(* CODESYS project Mahle_FilterLine_TempControl_02_08_20.project
   Title: Mahle_FilterLine_TempControl_03_01_20
   Version: 0.0.0.0

Project tree, tasks and I/O mapping:
  MyController : TM218LDAE24DRHN, Schneider Electric, order no. TM218LDAE24DRHN, version 4.0.1.26
      settings: Expansion Tasks.Expansion 1 Task Name = 'MAST'; Expansion Tasks.Expansion 2 Task Name = 'MAST'
    application Application
      libraries: Standard, * (System)
      task MAST (cyclic, interval 20 ms, priority 15, watchdog 100 ms x 1) calls POU, POU_MC2
      function HiddenPOU [ST]
      global variables GVL
      program POU [FBD]
      function block tempAvergaging [ST]
      function block tempController [ST]
      function block calculateCycleTime [ST]
      function CheckBounds [ST]
      function block pressureAlarm [ST]
      program POU_MC2 [FBD]
    Embedded Functions
      IO : IO, Schneider Electric, version 4.0.1.26
          input  iwIO_IW0 : WORD  // IW0
          input  iAuto : BOOL  // IW0.I0
          input  iThyristorTrip2 : BOOL  // IW0.I1
          input  iStartPB : BOOL  // IW0.I2
          input  iStopPB : BOOL  // IW0.I3
          input  iStartPB2 : BOOL  // IW0.I4
          input  iStopPB2 : BOOL  // IW0.I5
          input  iThyristorTrip : BOOL  // IW0.I6
          input  iFwdSensor2 : BOOL  // IW0.I7
          input  iFwdSensor : BOOL  // IW0.I8
          input  iSafetyGuard : BOOL  // IW0.I10
          input  iSafetyGuard2 : BOOL  // IW0.I11
          input  iPanelPB : BOOL  // IW0.I13
          output qStartMC : BOOL  // QW0.Q0
          output qHeaterDown : BOOL  // QW0.Q1
          output qYellow : BOOL  // QW0.Q2
          output qGreen : BOOL  // QW0.Q3
          output qRed : BOOL  // QW0.Q4
          output qHooter : BOOL  // QW0.Q5
          output qStopCmd : BOOL  // QW0.Q6
          output qHeaterDown2 : BOOL  // QW0.Q7
          output qStartMC2 : BOOL  // QW0.Q8
          output qStopCmd2 : BOOL  // QW0.Q9
          unmapped channels: QW0
      HSC : HSC, Schneider Electric, version 4.0.1.26
    Serial Line 1
      SoMachine_Network_Manager : SoMachine-Network Manager, Schneider Electric, version 4.0.0.2
    Serial Line 2
      Modbus_Manager : Modbus Manager, Schneider Electric, version 4.0.0.2
    Ethernet
        settings: IPAddress = [192, 168, 1, 1]; SubnetMask = [255, 255, 255, 0]; GatewayAddress = [192, 168, 1, 1]; WebServer = FALSE; FTP Server = FALSE; SoMachine Protocol = TRUE; Modbus Server = TRUE; NetManage Protocol = FALSE; SNMP protocol = FALSE; Enable Routing = FALSE
    Module_1 : TM2AMM3HT, Schneider Electric, order no. TM2AMM3HT, version 4.0.1.26
        settings: IW0.Maximum = 4000; IW1.Maximum = 1000; QW0.Maximum = 1000
        input  iwTempSensor : INT  // IW0
        input  iwPressureSensor : INT  // IW1
        output qwHeater : INT  // QW0
    Module_2 : TM2AMM3HT, Schneider Electric, order no. TM2AMM3HT, version 4.0.1.26
        settings: IW0.Maximum = 4000; IW1.Maximum = 1000; QW0.Maximum = 1000
        input  iwTempSensor2 : INT  // IW0
        input  iwPressureSensor2 : INT  // IW1
        output qwHeater2 : INT  // QW0
*)

// MyController/Application/GVL
VAR_GLOBAL
	thyristorTrip AT %MX600.0: BOOL;
	autoSel AT %MX600.1: BOOL;
	mcRunning AT %MX600.2: BOOL;
	heaterDown AT %MX600.3: BOOL;
	startSensing AT %MX600.4: BOOL;
	pressureLow AT %MX600.5: BOOL;
	resetPressMinMax AT %MX600.6: BOOL;
	cycleError AT %MX600.7: BOOL;
	startMCRun: BOOL;
	
	pressLowAlarm: BOOL;
	pressHighAlarm: BOOL;
	
	//MC2
	thyristorTrip2 AT %MX610.0: BOOL;
	autoSel2 AT %MX610.1: BOOL;
	mcRunning2 AT %MX610.2: BOOL;
	heaterDown2 AT %MX610.3: BOOL;
	startSensing2 AT %MX610.4: BOOL;
	pressureLow2 AT %MX610.5: BOOL;
	resetPressMinMax2 AT %MX610.6: BOOL;
	cycleError2 AT %MX610.7: BOOL;
	startMCRun2: BOOL;
	
	pressLowAlarm2: BOOL;
	pressHighAlarm2: BOOL;
	
	green2: BOOL;
	yellow2: BOOL;
	red2: BOOL;
END_VAR
VAR_GLOBAL RETAIN
	tempOffset AT %MD0: REAL :=0;
	puckTemp AT %MD1: REAL;
	finalCount AT %MD2: DINT;
	propGain AT %MD3: REAL;
	integGain AT %MD4: REAL;
	derivative AT %MD5: REAL;
	setTemp AT %MD6: REAL :=195;
	puckTempAvg AT %MD7: REAL;
	heaterManualSP AT %MD8: REAL :=50;
	heaterPIDOut AT %MD9: REAL;
	
	cycleTime AT %MD10: REAL;
	timeBWPucks AT %MD11: REAL;
	heaterLowRun AT %MD12: REAL :=48;
	heaterHighRun AT %MD13: REAL :=55;
	
	pressure AT %MD14: REAL;
	pressHighSet AT %MD15: REAL;
	pressLowSet AT %MD16: REAL;
	pressMin AT %MD17: REAL;
	pressMax AT %MD18: REAL;	
	pressureOffset AT %MD19: REAL;
	AvgPressure AT %MD21: REAL;
	pressurePSI AT %MD22: REAL;
	
	startDelay AT %MW100: INT :=6;
	mcStopTime AT %MW101: INT :=30;
	pressAlarmDelay AT %MW102: INT;
	
	heaterManualOn AT %MX602.0: BOOL;
	heaterManualDown AT %MX602.1: BOOL;
	
	
	//MC2
	tempOffset2 AT %MD100: REAL :=0;
	puckTemp2 AT %MD101: REAL;
	finalCount2 AT %MD102: DINT;
	propGain2 AT %MD103: REAL;
	integGain2 AT %MD104: REAL;
	derivative2 AT %MD105: REAL;
	setTemp2 AT %MD106: REAL :=195;
	puckTempAvg2 AT %MD107: REAL;
	heaterManualSP2 AT %MD108: REAL :=50;
	heaterPIDOut2 AT %MD109: REAL;
	
	cycleTime2 AT %MD110: REAL;
	timeBWPucks2 AT %MD111: REAL;
	heaterLowRun2 AT %MD112: REAL :=48;
	heaterHighRun2 AT %MD113: REAL :=55;
	
	pressure2 AT %MD114: REAL;
	pressHighSet2 AT %MD115: REAL;
	pressLowSet2 AT %MD116: REAL;
	pressMin2 AT %MD117: REAL;
	pressMax2 AT %MD118: REAL;	
	pressureOffset2 AT %MD119: REAL;
	AvgPressure2 AT %MD121: REAL;
	pressurePSI2 AT %MD122: REAL;
	
	startDelay2 AT %MW110: INT :=6;
	mcStopTime2 AT %MW111: INT :=30;
	pressAlarmDelay2 AT %MW112: INT;
	
	heaterManualOn2 AT %MX612.0: BOOL;
	heaterManualDown2 AT %MX612.1: BOOL;
	
END_VAR

// MyController/Application/POU
PROGRAM POU
VAR
	puckTemp1: REAL;
	tempAvergaging_0: tempAvergaging;
	PID_0: PID;
	RS_0: RS;
	runMC: BOOL;
	R_TRIG_0: R_TRIG;
	PID_1: PID_FIXCYCLE;
	TON_0: TON;
	tempController_0: tempController;
	TP_0: TP;
	mcStartDelayTime: TIME;
	TON_1: TON;
	calculateCycleTime_0: calculateCycleTime;
	sensorTrig: BOOL;
	TP_1: TP;
	stopTime: TIME;
	TON_2: TON;
	stopTimeET: TIME;
	stopHeater: BOOL;
	pressureAlarm_0: pressureAlarm;
	pressAlarm: BOOL;
	startProduction: BOOL;
	greenCont: BOOL;
	BLINK_0: BLINK;
	BLINK_1: BLINK;
	stopHeater1: BOOL;
	RS_1: RS;
	R_TRIG_1: R_TRIG;
	R_TRIG_2: R_TRIG;
	R_TRIG_3: R_TRIG;
	R_TRIG_4: R_TRIG;
	RS_2: RS;
	stopMC: BOOL;
	BLINK_2: BLINK;
	stopCommand: BOOL;
	CTU_0: CTU;
	R_TRIG_5: R_TRIG;
	TON_3: TON;
END_VAR

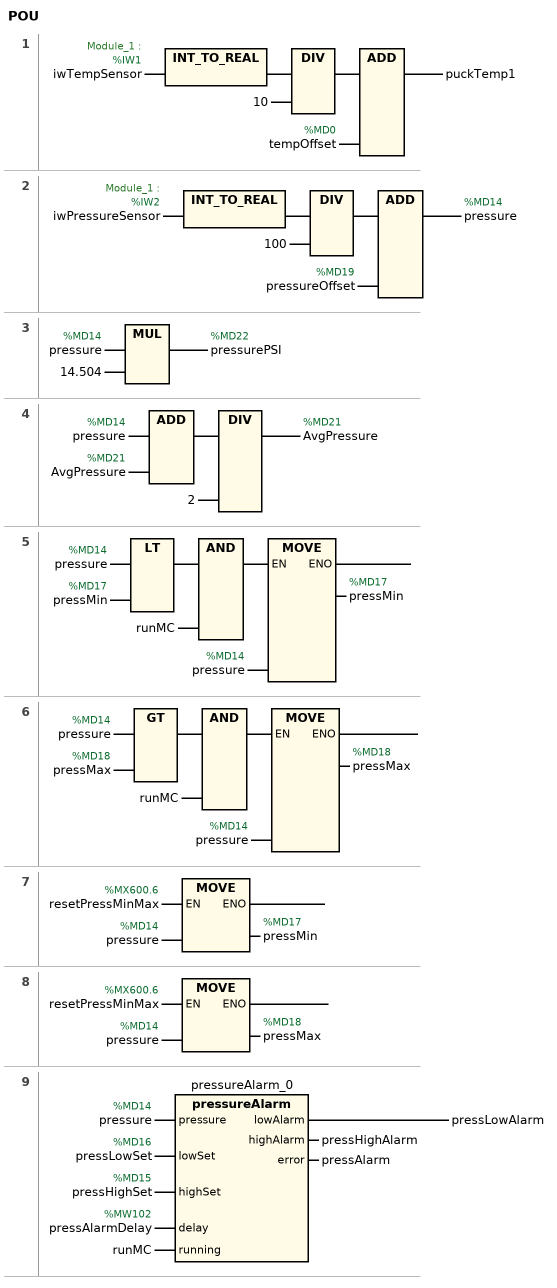
// NETWORK 1
//   iwTempSensor: Module_1 : | AT %IW1
//   tempOffset: AT %MD0
puckTemp1 := INT_TO_REAL(iwTempSensor) / 10 + tempOffset;

// NETWORK 2
//   iwPressureSensor: Module_1 : | AT %IW2
//   pressureOffset: AT %MD19
//   pressure: AT %MD14
pressure := INT_TO_REAL(iwPressureSensor) / 100 + pressureOffset;

// NETWORK 3
//   pressure: AT %MD14
//   pressurePSI: AT %MD22
pressurePSI := pressure * 14.504;

// NETWORK 4
//   pressure: AT %MD14
//   AvgPressure: AT %MD21
AvgPressure := (pressure + AvgPressure) / 2;

// NETWORK 5
//   pressure: AT %MD14
//   pressMin: AT %MD17
IF pressure < pressMin AND runMC THEN pressMin := pressure; END_IF

// NETWORK 6
//   pressure: AT %MD14
//   pressMax: AT %MD18
IF pressure > pressMax AND runMC THEN pressMax := pressure; END_IF

// NETWORK 7
//   resetPressMinMax: AT %MX600.6
//   pressure: AT %MD14
//   pressMin: AT %MD17
IF resetPressMinMax THEN pressMin := pressure; END_IF

// NETWORK 8
//   resetPressMinMax: AT %MX600.6
//   pressure: AT %MD14
//   pressMax: AT %MD18
IF resetPressMinMax THEN pressMax := pressure; END_IF

// NETWORK 9
//   pressure: AT %MD14
//   pressLowSet: AT %MD16
//   pressHighSet: AT %MD15
//   pressAlarmDelay: AT %MW102
pressureAlarm_0(
    pressure := pressure,
    lowSet := pressLowSet,
    highSet := pressHighSet,
    delay := pressAlarmDelay,
    running := runMC,
    highAlarm => pressHighAlarm,
    error => pressAlarm); // pressureAlarm
pressLowAlarm := pressureAlarm_0.lowAlarm;

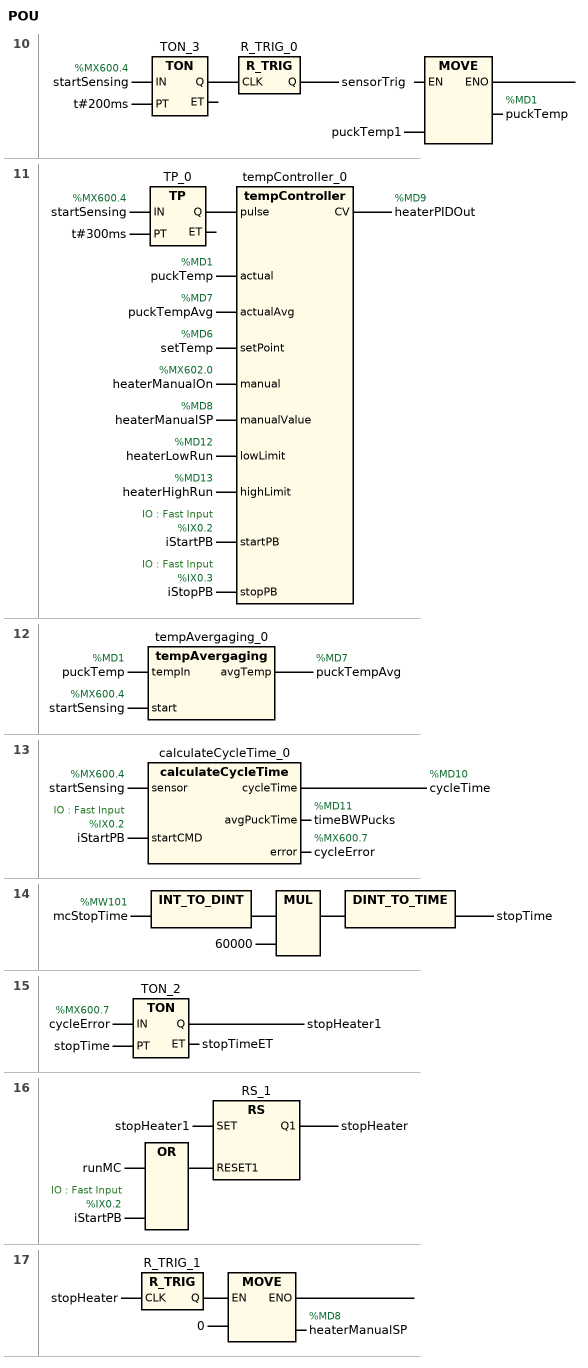
// NETWORK 10
//   startSensing: AT %MX600.4
//   puckTemp: AT %MD1
TON_3(IN := startSensing, PT := t#200ms); // TON
R_TRIG_0(CLK := TON_3.Q); // R_TRIG
sensorTrig := R_TRIG_0.Q;
IF R_TRIG_0.Q THEN puckTemp := puckTemp1; END_IF

// NETWORK 11
//   startSensing: AT %MX600.4
//   puckTemp: AT %MD1
//   puckTempAvg: AT %MD7
//   setTemp: AT %MD6
//   heaterManualOn: AT %MX602.0
//   heaterManualSP: AT %MD8
//   heaterLowRun: AT %MD12
//   heaterHighRun: AT %MD13
//   iStartPB: IO : Fast Input | AT %IX0.2
//   iStopPB: IO : Fast Input | AT %IX0.3
//   heaterPIDOut: AT %MD9
TP_0(IN := startSensing, PT := t#300ms); // TP
tempController_0(
    pulse := TP_0.Q,
    actual := puckTemp,
    actualAvg := puckTempAvg,
    setPoint := setTemp,
    manual := heaterManualOn,
    manualValue := heaterManualSP,
    lowLimit := heaterLowRun,
    highLimit := heaterHighRun,
    startPB := iStartPB,
    stopPB := iStopPB); // tempController
heaterPIDOut := tempController_0.CV;

// NETWORK 12
//   puckTemp: AT %MD1
//   startSensing: AT %MX600.4
//   puckTempAvg: AT %MD7
tempAvergaging_0(tempIn := puckTemp, start := startSensing); // tempAvergaging
puckTempAvg := tempAvergaging_0.avgTemp;

// NETWORK 13
//   startSensing: AT %MX600.4
//   iStartPB: IO : Fast Input | AT %IX0.2
//   timeBWPucks: AT %MD11
//   cycleError: AT %MX600.7
//   cycleTime: AT %MD10
calculateCycleTime_0(
    sensor := startSensing,
    startCMD := iStartPB,
    avgPuckTime => timeBWPucks,
    error => cycleError); // calculateCycleTime
cycleTime := calculateCycleTime_0.cycleTime;

// NETWORK 14
//   mcStopTime: AT %MW101
stopTime := DINT_TO_TIME(INT_TO_DINT(mcStopTime) * 60000);

// NETWORK 15
//   cycleError: AT %MX600.7
TON_2(IN := cycleError, PT := stopTime, ET => stopTimeET); // TON
stopHeater1 := TON_2.Q;

// NETWORK 16
//   iStartPB: IO : Fast Input | AT %IX0.2
RS_1(SET := stopHeater1, RESET1 := runMC OR iStartPB); // RS
stopHeater := RS_1.Q1;

// NETWORK 17
//   heaterManualSP: AT %MD8
R_TRIG_1(CLK := stopHeater); // R_TRIG
IF R_TRIG_1.Q THEN heaterManualSP := 0; END_IF

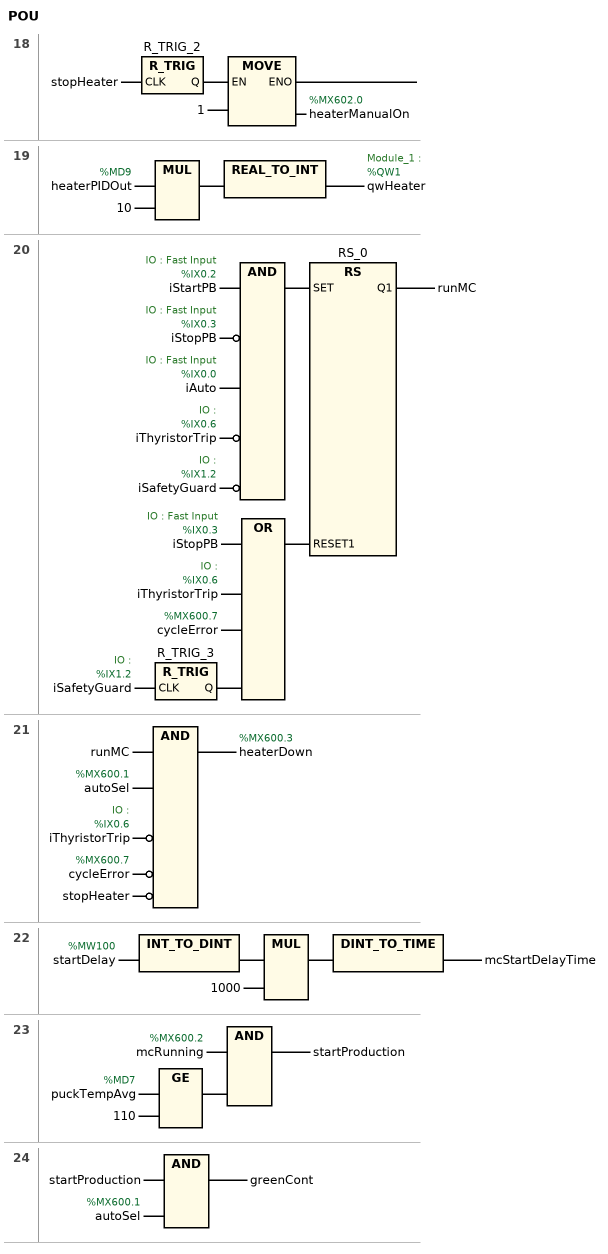
// NETWORK 18
//   heaterManualOn: AT %MX602.0
R_TRIG_2(CLK := stopHeater); // R_TRIG
IF R_TRIG_2.Q THEN heaterManualOn := 1; END_IF

// NETWORK 19
//   heaterPIDOut: AT %MD9
//   qwHeater: Module_1 : | AT %QW1
qwHeater := REAL_TO_INT(heaterPIDOut * 10);

// NETWORK 20
//   iStartPB: IO : Fast Input | AT %IX0.2
//   iStopPB: IO : Fast Input | AT %IX0.3
//   iAuto: IO : Fast Input | AT %IX0.0
//   iThyristorTrip: IO : | AT %IX0.6
//   iSafetyGuard: IO : | AT %IX1.2
//   cycleError: AT %MX600.7
R_TRIG_3(CLK := iSafetyGuard); // R_TRIG
RS_0(SET := iStartPB AND NOT iStopPB AND iAuto AND NOT iThyristorTrip AND NOT iSafetyGuard, RESET1 := iStopPB OR iThyristorTrip OR cycleError OR R_TRIG_3.Q); // RS
runMC := RS_0.Q1;

// NETWORK 21
//   autoSel: AT %MX600.1
//   iThyristorTrip: IO : | AT %IX0.6
//   cycleError: AT %MX600.7
//   heaterDown: AT %MX600.3
heaterDown := runMC AND autoSel AND NOT iThyristorTrip AND NOT cycleError AND NOT stopHeater;

// NETWORK 22
//   startDelay: AT %MW100
mcStartDelayTime := DINT_TO_TIME(INT_TO_DINT(startDelay) * 1000);

// NETWORK 23
//   mcRunning: AT %MX600.2
//   puckTempAvg: AT %MD7
startProduction := mcRunning AND puckTempAvg >= 110;

// NETWORK 24
//   autoSel: AT %MX600.1
greenCont := startProduction AND autoSel;

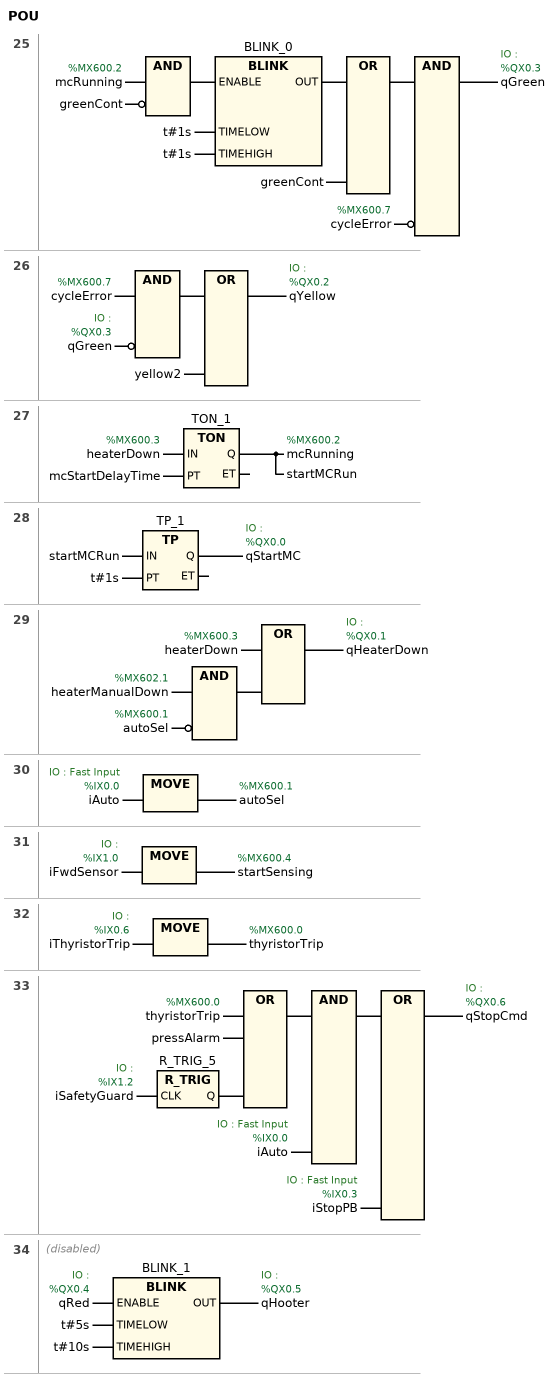
// NETWORK 25
//   mcRunning: AT %MX600.2
//   cycleError: AT %MX600.7
//   qGreen: IO : | AT %QX0.3
BLINK_0(ENABLE := mcRunning AND NOT greenCont, TIMELOW := t#1s, TIMEHIGH := t#1s); // BLINK
qGreen := (BLINK_0.OUT OR greenCont) AND NOT cycleError;

// NETWORK 26
//   cycleError: AT %MX600.7
//   qGreen: IO : | AT %QX0.3
//   qYellow: IO : | AT %QX0.2
qYellow := cycleError AND NOT qGreen OR yellow2;

// NETWORK 27
//   heaterDown: AT %MX600.3
//   mcRunning: AT %MX600.2
TON_1(IN := heaterDown, PT := mcStartDelayTime); // TON
mcRunning := TON_1.Q;
startMCRun := TON_1.Q;

// NETWORK 28
//   qStartMC: IO : | AT %QX0.0
TP_1(IN := startMCRun, PT := t#1s); // TP
qStartMC := TP_1.Q;

// NETWORK 29
//   heaterDown: AT %MX600.3
//   heaterManualDown: AT %MX602.1
//   autoSel: AT %MX600.1
//   qHeaterDown: IO : | AT %QX0.1
qHeaterDown := heaterDown OR heaterManualDown AND NOT autoSel;

// NETWORK 30
//   iAuto: IO : Fast Input | AT %IX0.0
//   autoSel: AT %MX600.1
autoSel := iAuto;

// NETWORK 31
//   iFwdSensor: IO : | AT %IX1.0
//   startSensing: AT %MX600.4
startSensing := iFwdSensor;

// NETWORK 32
//   iThyristorTrip: IO : | AT %IX0.6
//   thyristorTrip: AT %MX600.0
thyristorTrip := iThyristorTrip;

// NETWORK 33
//   thyristorTrip: AT %MX600.0
//   iSafetyGuard: IO : | AT %IX1.2
//   iAuto: IO : Fast Input | AT %IX0.0
//   iStopPB: IO : Fast Input | AT %IX0.3
//   qStopCmd: IO : | AT %QX0.6
R_TRIG_5(CLK := iSafetyGuard); // R_TRIG
qStopCmd := (thyristorTrip OR pressAlarm OR R_TRIG_5.Q) AND iAuto OR iStopPB;

// NETWORK 34 (disabled)
//   qRed: IO : | AT %QX0.4
//   qHooter: IO : | AT %QX0.5
// BLINK_1(ENABLE := qRed, TIMELOW := t#5s, TIMEHIGH := t#10s); // BLINK
// qHooter := BLINK_1.OUT;

END_PROGRAM

// MyController/Application/pressureAlarm
FUNCTION_BLOCK pressureAlarm
VAR_INPUT
	pressure: REAL;
	lowSet: REAL;
	highSet: REAL;
	delay: INT;
	running: BOOL;
END_VAR
VAR_OUTPUT
	lowAlarm: BOOL;
	highAlarm: BOOL;
	error: BOOL;
END_VAR
VAR
	timeDelay: TIME;
	startTON1: BOOL;
	startTON2: BOOL;
	TON1: TON;
	TON2: TON;
END_VAR

timeDelay := DINT_TO_TIME(INT_TO_DINT(delay)*1000);

TON1(IN:=startTON1, PT:=timeDelay);
TON2(IN:=startTON2, PT:=timeDelay);

IF running THEN
	IF pressure < lowSet THEN
		startTON1 := TRUE;
	ELSE
		startTON1 := FALSE;
	END_IF

	IF pressure > highSet THEN
		startTON2 := TRUE;
	ELSE
		startTON2 := FALSE;
	END_IF			
	
	IF ton1.Q THEN
		lowAlarm := TRUE;
	ELSE
		lowAlarm := FALSE;
	END_IF
	
	IF ton2.Q THEN
		highAlarm := TRUE;
	ELSE
		highAlarm := FALSE;
	END_IF
	
	IF lowAlarm OR highAlarm THEN
		error := TRUE;
	ELSE
		error := FALSE;
	END_IF
ELSE
	lowAlarm := FALSE;
	highAlarm := FALSE;
	error := false;
END_IF

END_FUNCTION_BLOCK

// MyController/Application/tempController
FUNCTION_BLOCK tempController
VAR_INPUT
	pulse: BOOL;
	actual: REAL;
	actualAvg: REAL;
	setPoint: REAL;
	manual: BOOL;
	manualValue: REAL;
	lowLimit: REAL;
	highLimit: REAL;
	startPB: BOOL;
	stopPB: BOOL;
END_VAR
VAR_OUTPUT
	CV: REAL;
END_VAR
VAR
	error: REAL;
	errorPC: REAL;
	CV1: REAL;
	errorPCAbs: REAL;
	errorFromAvg: REAL;
	startHeater: BOOL;
	CV2: REAL;
END_VAR

IF startPB AND NOT manual THEN
	startHeater := TRUE;
	CV1 := highLimit;
END_IF
IF pulse AND NOT manual THEN
	error := setPoint - actual;
	errorPC := (error*100)/setPoint;
	errorFromAvg := actualAvg - actual;
	IF errorFromAvg < 20 AND errorFromAvg > -20 THEN
	
		IF errorPC >=0 THEN
			errorPCAbs := errorPC;
		ELSE
			errorPCAbs := -1*errorPC;
		END_IF
	
		IF errorPCAbs < 2 THEN
			CV1 := CV+(errorPC/90);
		ELSIF errorPCAbs < 5 THEN
			CV1 := CV + (errorPC/50);
		ELSIF errorPCAbs < 15 THEN
			CV1 := CV + (errorPC/75);
		ELSE
			CV1 := CV + (errorPC/100);				
		END_IF
	END_IF
END_IF

IF manual THEN
	CV := manualValue;
ELSE
	CV := CV2;
END_IF

IF CV1 < lowLimit THEN
	CV2 := lowLimit;
ELSIF CV1 > highLimit THEN
	CV2 := highLimit;
ELSE
	CV2 := CV1;
END_IF

END_FUNCTION_BLOCK

// MyController/Application/tempAvergaging
FUNCTION_BLOCK tempAvergaging
VAR_INPUT
	tempIn: REAL;
	start: BOOL;
END_VAR
VAR_OUTPUT
	avgTemp: REAL;
END_VAR
VAR
	counter1: CTU;
	x1: REAL :=0;
	x2: REAL :=0;
	x3: REAL :=0;
	x4: REAL :=0;
	x5: REAL :=0;
	x6: REAL :=0;
	x7: REAL :=0;
	x8: REAL :=0;
	x9: REAL :=0;
	x10: REAL :=0;
	x11: REAL :=0;
	x12: REAL :=0;
	countReset: BOOL;
END_VAR

counter1(CU:=start, RESET:=countReset, PV:=5);
CASE counter1.CV OF
	1:	x1:=tempIn;
	2:	x2:=tempIn;
	3:	x3:=tempIn;
	4:	x4:=tempIn;
	5:	x5:=tempIn;
//	6:	x6:=tempIn;
//	7:	x7:=tempIn;
//	8:	x8:=tempIn;
//	9:	x9:=tempIn;
//	10:	x10:=tempIn;
//	11:	x11:=tempIn;
//	12:	x12:=tempIn;
END_CASE

IF counter1.Q THEN
	countReset := TRUE;
ELSE
	countReset := FALSE;
END_IF

//avgTemp := (x1+x2+x3+x4+x5+x6+x7+x8+x9+x10+x11+x12)/12;

avgTemp := (x1+x2+x3+x4+x5)/5;

END_FUNCTION_BLOCK

// MyController/Application/calculateCycleTime
FUNCTION_BLOCK calculateCycleTime
VAR_INPUT
	sensor: BOOL;
	startCMD: BOOL;
END_VAR
VAR_OUTPUT
	cycleTime: REAL;
	avgPuckTime: REAL;
	error: BOOL;
END_VAR
VAR
	ton1: TON;
	ton2: TON;
	ton3: TON;
	ctu1: CTU;
	ctu2: CTU;
	ctuReset: BOOL;
	startTON1: BOOL;
	startTON2: BOOL;
	startTON3: BOOL;
	startTON4: BOOL;
	t1Time: REAL;
	t2Time: REAL;
	t3Time: REAL;
	t4Time: REAL;
	ctuReset2: BOOL;
	t1: REAL;
	t2: REAL;
	t3: REAL;
	t4: REAL;
	t5: REAL;
	t6: REAL;
	t7: REAL;
	t8: REAL;
	t9: REAL;
	t10: REAL;
	t11: REAL;
	t12: REAL;
	t13: REAL;
	t14: REAL;
	t15: REAL;
	t16: REAL;
	t17: REAL;
	t18: REAL;
	t19: REAL;
	t20: REAL;
	t21: REAL;
	t22: REAL;
	t23: REAL;
	t24: REAL;
	firstRun: BOOL;
	ton4: TON;
	ton5: TON;
	newCycleStart: BOOL;
	rtrig1: R_TRIG;
	rtrig2: R_TRIG;
	trig2: BOOL;
	t1TimeInit: REAL;
	t2TimeInit: REAL;
	ctu3: CTU;
	cycleDone: BOOL;
	ctu3Reset: BOOL;
	t4TimeInit: REAL;
	t3TimeInit: REAL;
	tof1: TOF;
END_VAR

ctu1(CU:=sensor, RESET:=ctuReset, PV:=2);
ton1(IN:=startTON1, PT:=T#30M);
ton2(IN:=startTON2, PT:=T#30M);
ton3(IN:=startTON3, PT:=T#60M);
ton4(IN:=startTON4, PT:=T#60M);
ton5(IN:=newCycleStart, PT:=T#100MS);
ctu2(CU:=sensor, RESET:=ctu2.Q, PV:=2);
ctu3(CU:=cycleDone, RESET:=ctu3Reset, PV:=2);
tof1(IN:=startCMD, PT:=T#10S);

	IF ctu1.CV = 1 AND NOT error THEN
		startTON1 := TRUE;
		startTON2:= FALSE;	
		t2Time := t2TimeInit;
	END_IF

	IF ctu1.CV = 2 AND NOT error THEN
		startTON1:=FALSE;
		startTON2:= TRUE;
		t1Time := t1TimeInit;
	END_IF
	
	IF startCMD THEN
		ctuReset := TRUE;
	END_IF
	
	IF ctu1.CV >= 2 THEN
		ctuReset := TRUE;
	ELSE	
		ctuReset := FALSE;
	END_IF

	IF startTON1 THEN
		t1TimeInit := TIME_TO_REAL(ton1.ET);
	END_IF

	IF startTON2 THEN
		t2TimeInit := TIME_TO_REAL(ton2.ET);
	END_IF

	CASE ctu2.CV OF
		0:	t1:=t2Time;
		1:	t2:=t1Time;
		2:	t3:=t2Time;
		3:	t4:=t1Time;
		4:	t5:=t2Time;
		5:	t6:=t1Time;
		6:	t7:=t2Time;
		7:	t8:=t1Time;
		8:	t9:=t2Time;
		9:	t10:=t1Time;
		10:	t11:=t2Time;
		11:	t12:=t1Time;
		12:	t13:=t2Time;
		13:	t14:=t1Time;
		14:	t15:=t2Time;
		15:	t16:=t1Time;
		16:	t17:=t2Time;
		17:	t18:=t1Time;
		18:	t19:=t2Time;
		19:	t20:=t1Time;
		20:	t21:=t2Time;
		21:	t22:=t1Time;
		22:	t23:=t2Time;
		23:	t24:=t1Time;
		
	END_CASE
		
	IF TIME_TO_REAL(ton1.ET) > MIN((avgPuckTime*1000+2000),8000) AND NOT tof1.Q THEN
		error := TRUE;
	ELSIF TIME_TO_REAL(ton2.ET) > MIN((avgPuckTime*1000+2000),8000)  AND NOT tof1.Q THEN
		error := TRUE;
	ELSE
		error := FALSE;
	END_IF
	
	IF startTON3 THEN
		t3TimeInit := TIME_TO_REAL(ton3.ET);
	END_IF
	IF startTON4 THEN
		t4TimeInit := TIME_TO_REAL(ton4.ET);
	END_IF

	IF ctu2.CV = 1 THEN
		cycleDone := TRUE;
	ELSE
		cycleDone := FALSE;
	END_IF
	
	IF ctu3.CV = 1 THEN
		startTON3 := TRUE;
		startTON4:= FALSE;	
		t4Time := t4TimeInit;
	END_IF

	IF ctu3.CV = 2 THEN
		startTON3:=FALSE;
		startTON4:= TRUE;
		t3Time := t3TimeInit;
	END_IF
	
	IF ctu3.CV >= 2 THEN
		ctu3Reset := TRUE;
	ELSE	
		ctu3Reset := FALSE;
	END_IF
	
	IF NOT error THEN
		//avgPuckTime := (t1+t2+t3+t4+t5+t6+t7+t8+t9+t10+t11+t12+t13+t14+t15+t16+t17+t18+t19+t20+t21+t22+t23+t24)/24000;
		avgPuckTime := (t1+t2)/2000;
		cycleTime := (t3Time+t4Time)/2000;
	END_IF

END_FUNCTION_BLOCK

// MyController/Application/POU_MC2
PROGRAM POU_MC2
VAR
	puckTemp1: REAL;
	tempAvergaging_0: tempAvergaging;
	PID_0: PID;
	RS_0: RS;
	runMC: BOOL;
	R_TRIG_0: R_TRIG;
	PID_1: PID_FIXCYCLE;
	TON_0: TON;
	tempController_0: tempController;
	TP_0: TP;
	mcStartDelayTime: TIME;
	TON_1: TON;
	calculateCycleTime_0: calculateCycleTime;
	sensorTrig: BOOL;
	TP_1: TP;
	stopTime: TIME;
	TON_2: TON;
	stopTimeET: TIME;
	stopHeater: BOOL;
	pressureAlarm_0: pressureAlarm;
	pressAlarm: BOOL;
	startProduction: BOOL;
	greenCont: BOOL;
	BLINK_0: BLINK;
	BLINK_1: BLINK;
	stopHeater1: BOOL;
	RS_1: RS;
	R_TRIG_1: R_TRIG;
	R_TRIG_2: R_TRIG;
	R_TRIG_3: R_TRIG;
	R_TRIG_4: R_TRIG;
	RS_2: RS;
	stopMC: BOOL;
	BLINK_2: BLINK;
	stopCommand: BOOL;
	CTU_0: CTU;
	R_TRIG_5: R_TRIG;
	TON_3: TON;
END_VAR

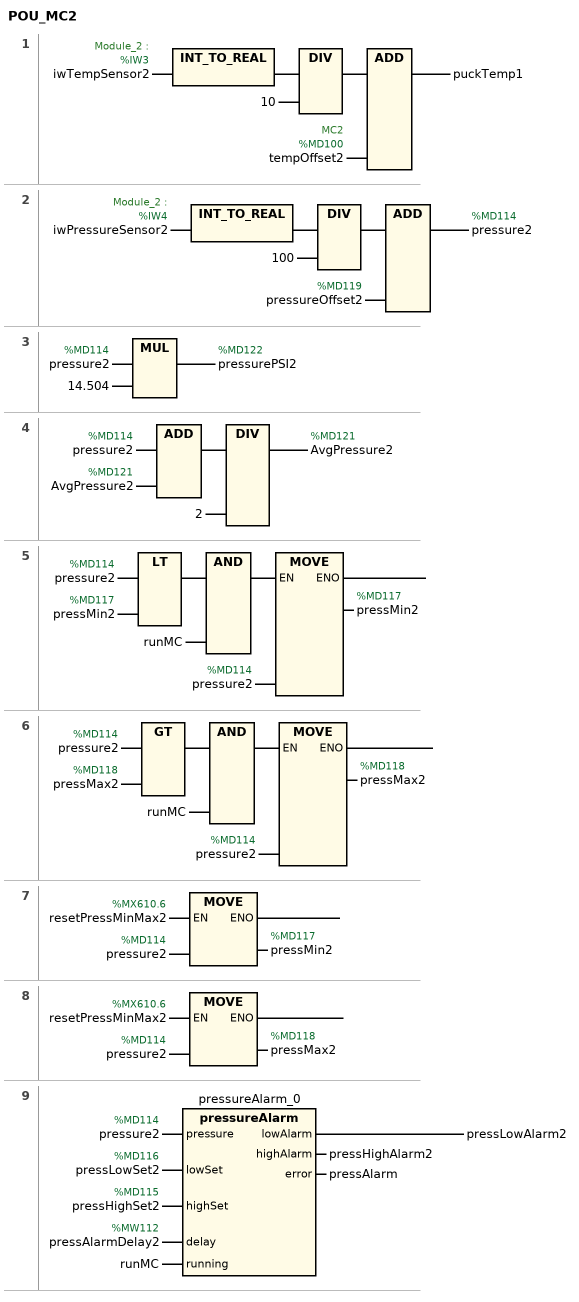
// NETWORK 1
//   iwTempSensor2: Module_2 : | AT %IW3
//   tempOffset2: MC2 | AT %MD100
puckTemp1 := INT_TO_REAL(iwTempSensor2) / 10 + tempOffset2;

// NETWORK 2
//   iwPressureSensor2: Module_2 : | AT %IW4
//   pressureOffset2: AT %MD119
//   pressure2: AT %MD114
pressure2 := INT_TO_REAL(iwPressureSensor2) / 100 + pressureOffset2;

// NETWORK 3
//   pressure2: AT %MD114
//   pressurePSI2: AT %MD122
pressurePSI2 := pressure2 * 14.504;

// NETWORK 4
//   pressure2: AT %MD114
//   AvgPressure2: AT %MD121
AvgPressure2 := (pressure2 + AvgPressure2) / 2;

// NETWORK 5
//   pressure2: AT %MD114
//   pressMin2: AT %MD117
IF pressure2 < pressMin2 AND runMC THEN pressMin2 := pressure2; END_IF

// NETWORK 6
//   pressure2: AT %MD114
//   pressMax2: AT %MD118
IF pressure2 > pressMax2 AND runMC THEN pressMax2 := pressure2; END_IF

// NETWORK 7
//   resetPressMinMax2: AT %MX610.6
//   pressure2: AT %MD114
//   pressMin2: AT %MD117
IF resetPressMinMax2 THEN pressMin2 := pressure2; END_IF

// NETWORK 8
//   resetPressMinMax2: AT %MX610.6
//   pressure2: AT %MD114
//   pressMax2: AT %MD118
IF resetPressMinMax2 THEN pressMax2 := pressure2; END_IF

// NETWORK 9
//   pressure2: AT %MD114
//   pressLowSet2: AT %MD116
//   pressHighSet2: AT %MD115
//   pressAlarmDelay2: AT %MW112
pressureAlarm_0(
    pressure := pressure2,
    lowSet := pressLowSet2,
    highSet := pressHighSet2,
    delay := pressAlarmDelay2,
    running := runMC,
    highAlarm => pressHighAlarm2,
    error => pressAlarm); // pressureAlarm
pressLowAlarm2 := pressureAlarm_0.lowAlarm;

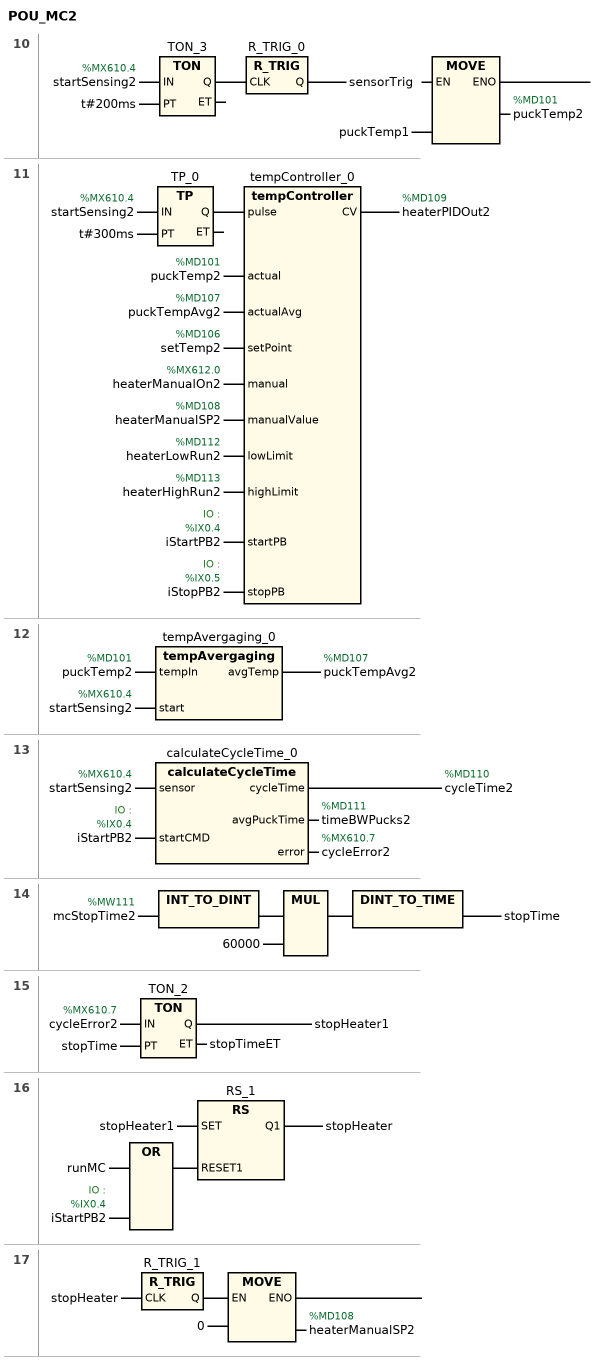
// NETWORK 10
//   startSensing2: AT %MX610.4
//   puckTemp2: AT %MD101
TON_3(IN := startSensing2, PT := t#200ms); // TON
R_TRIG_0(CLK := TON_3.Q); // R_TRIG
sensorTrig := R_TRIG_0.Q;
IF R_TRIG_0.Q THEN puckTemp2 := puckTemp1; END_IF

// NETWORK 11
//   startSensing2: AT %MX610.4
//   puckTemp2: AT %MD101
//   puckTempAvg2: AT %MD107
//   setTemp2: AT %MD106
//   heaterManualOn2: AT %MX612.0
//   heaterManualSP2: AT %MD108
//   heaterLowRun2: AT %MD112
//   heaterHighRun2: AT %MD113
//   iStartPB2: IO : | AT %IX0.4
//   iStopPB2: IO : | AT %IX0.5
//   heaterPIDOut2: AT %MD109
TP_0(IN := startSensing2, PT := t#300ms); // TP
tempController_0(
    pulse := TP_0.Q,
    actual := puckTemp2,
    actualAvg := puckTempAvg2,
    setPoint := setTemp2,
    manual := heaterManualOn2,
    manualValue := heaterManualSP2,
    lowLimit := heaterLowRun2,
    highLimit := heaterHighRun2,
    startPB := iStartPB2,
    stopPB := iStopPB2); // tempController
heaterPIDOut2 := tempController_0.CV;

// NETWORK 12
//   puckTemp2: AT %MD101
//   startSensing2: AT %MX610.4
//   puckTempAvg2: AT %MD107
tempAvergaging_0(tempIn := puckTemp2, start := startSensing2); // tempAvergaging
puckTempAvg2 := tempAvergaging_0.avgTemp;

// NETWORK 13
//   startSensing2: AT %MX610.4
//   iStartPB2: IO : | AT %IX0.4
//   timeBWPucks2: AT %MD111
//   cycleError2: AT %MX610.7
//   cycleTime2: AT %MD110
calculateCycleTime_0(
    sensor := startSensing2,
    startCMD := iStartPB2,
    avgPuckTime => timeBWPucks2,
    error => cycleError2); // calculateCycleTime
cycleTime2 := calculateCycleTime_0.cycleTime;

// NETWORK 14
//   mcStopTime2: AT %MW111
stopTime := DINT_TO_TIME(INT_TO_DINT(mcStopTime2) * 60000);

// NETWORK 15
//   cycleError2: AT %MX610.7
TON_2(IN := cycleError2, PT := stopTime, ET => stopTimeET); // TON
stopHeater1 := TON_2.Q;

// NETWORK 16
//   iStartPB2: IO : | AT %IX0.4
RS_1(SET := stopHeater1, RESET1 := runMC OR iStartPB2); // RS
stopHeater := RS_1.Q1;

// NETWORK 17
//   heaterManualSP2: AT %MD108
R_TRIG_1(CLK := stopHeater); // R_TRIG
IF R_TRIG_1.Q THEN heaterManualSP2 := 0; END_IF

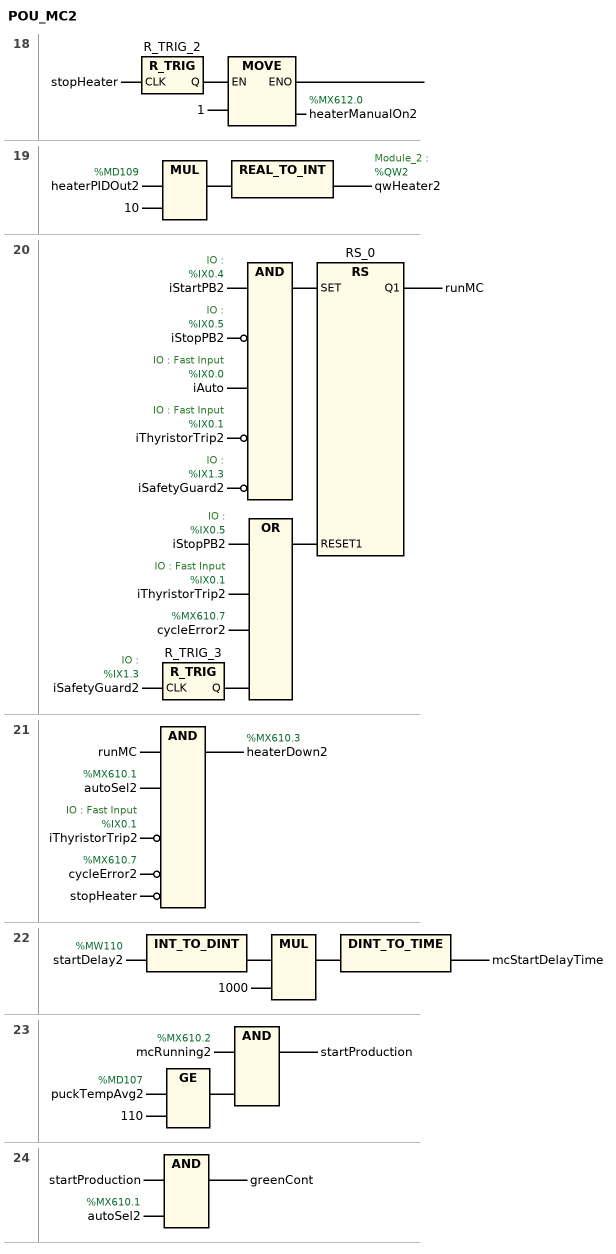
// NETWORK 18
//   heaterManualOn2: AT %MX612.0
R_TRIG_2(CLK := stopHeater); // R_TRIG
IF R_TRIG_2.Q THEN heaterManualOn2 := 1; END_IF

// NETWORK 19
//   heaterPIDOut2: AT %MD109
//   qwHeater2: Module_2 : | AT %QW2
qwHeater2 := REAL_TO_INT(heaterPIDOut2 * 10);

// NETWORK 20
//   iStartPB2: IO : | AT %IX0.4
//   iStopPB2: IO : | AT %IX0.5
//   iAuto: IO : Fast Input | AT %IX0.0
//   iThyristorTrip2: IO : Fast Input | AT %IX0.1
//   iSafetyGuard2: IO : | AT %IX1.3
//   cycleError2: AT %MX610.7
R_TRIG_3(CLK := iSafetyGuard2); // R_TRIG
RS_0(SET := iStartPB2 AND NOT iStopPB2 AND iAuto AND NOT iThyristorTrip2 AND NOT iSafetyGuard2, RESET1 := iStopPB2 OR iThyristorTrip2 OR cycleError2 OR R_TRIG_3.Q); // RS
runMC := RS_0.Q1;

// NETWORK 21
//   autoSel2: AT %MX610.1
//   iThyristorTrip2: IO : Fast Input | AT %IX0.1
//   cycleError2: AT %MX610.7
//   heaterDown2: AT %MX610.3
heaterDown2 := runMC AND autoSel2 AND NOT iThyristorTrip2 AND NOT cycleError2 AND NOT stopHeater;

// NETWORK 22
//   startDelay2: AT %MW110
mcStartDelayTime := DINT_TO_TIME(INT_TO_DINT(startDelay2) * 1000);

// NETWORK 23
//   mcRunning2: AT %MX610.2
//   puckTempAvg2: AT %MD107
startProduction := mcRunning2 AND puckTempAvg2 >= 110;

// NETWORK 24
//   autoSel2: AT %MX610.1
greenCont := startProduction AND autoSel2;

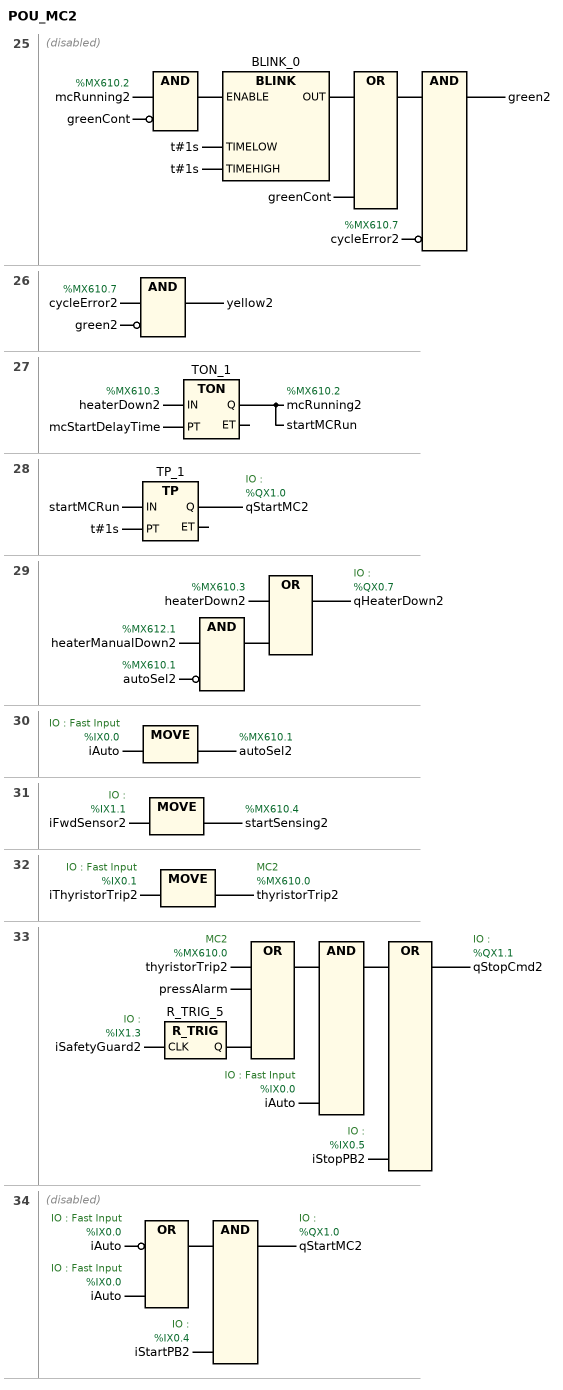
// NETWORK 25 (disabled)
//   mcRunning2: AT %MX610.2
//   cycleError2: AT %MX610.7
// BLINK_0(ENABLE := mcRunning2 AND NOT greenCont, TIMELOW := t#1s, TIMEHIGH := t#1s); // BLINK
// green2 := (BLINK_0.OUT OR greenCont) AND NOT cycleError2;

// NETWORK 26
//   cycleError2: AT %MX610.7
yellow2 := cycleError2 AND NOT green2;

// NETWORK 27
//   heaterDown2: AT %MX610.3
//   mcRunning2: AT %MX610.2
TON_1(IN := heaterDown2, PT := mcStartDelayTime); // TON
mcRunning2 := TON_1.Q;
startMCRun := TON_1.Q;

// NETWORK 28
//   qStartMC2: IO : | AT %QX1.0
TP_1(IN := startMCRun, PT := t#1s); // TP
qStartMC2 := TP_1.Q;

// NETWORK 29
//   heaterDown2: AT %MX610.3
//   heaterManualDown2: AT %MX612.1
//   autoSel2: AT %MX610.1
//   qHeaterDown2: IO : | AT %QX0.7
qHeaterDown2 := heaterDown2 OR heaterManualDown2 AND NOT autoSel2;

// NETWORK 30
//   iAuto: IO : Fast Input | AT %IX0.0
//   autoSel2: AT %MX610.1
autoSel2 := iAuto;

// NETWORK 31
//   iFwdSensor2: IO : | AT %IX1.1
//   startSensing2: AT %MX610.4
startSensing2 := iFwdSensor2;

// NETWORK 32
//   iThyristorTrip2: IO : Fast Input | AT %IX0.1
//   thyristorTrip2: MC2 | AT %MX610.0
thyristorTrip2 := iThyristorTrip2;

// NETWORK 33
//   thyristorTrip2: MC2 | AT %MX610.0
//   iSafetyGuard2: IO : | AT %IX1.3
//   iAuto: IO : Fast Input | AT %IX0.0
//   iStopPB2: IO : | AT %IX0.5
//   qStopCmd2: IO : | AT %QX1.1
R_TRIG_5(CLK := iSafetyGuard2); // R_TRIG
qStopCmd2 := (thyristorTrip2 OR pressAlarm OR R_TRIG_5.Q) AND iAuto OR iStopPB2;

// NETWORK 34 (disabled)
//   iAuto: IO : Fast Input | AT %IX0.0
//   iStartPB2: IO : | AT %IX0.4
//   qStartMC2: IO : | AT %QX1.0
// qStartMC2 := (NOT iAuto OR iAuto) AND iStartPB2;

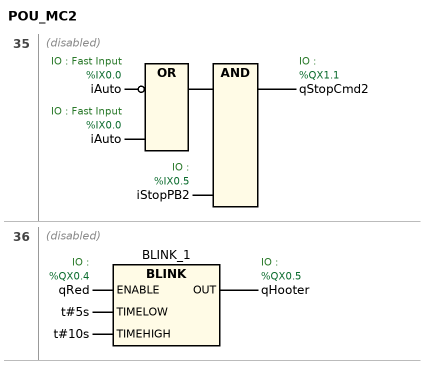
// NETWORK 35 (disabled)
//   iAuto: IO : Fast Input | AT %IX0.0
//   iStopPB2: IO : | AT %IX0.5
//   qStopCmd2: IO : | AT %QX1.1
// qStopCmd2 := (NOT iAuto OR iAuto) AND iStopPB2;

// NETWORK 36 (disabled)
//   qRed: IO : | AT %QX0.4
//   qHooter: IO : | AT %QX0.5
// BLINK_1(ENABLE := qRed, TIMELOW := t#5s, TIMEHIGH := t#10s); // BLINK
// qHooter := BLINK_1.OUT;

END_PROGRAM

// MyController/Application/HiddenPOU
FUNCTION HiddenPOU : BOOL

VAR_INPUT
	pHiddenFunc: POINTER TO WORD;
END_VAR
VAR
	pRead: POINTER TO BYTE;
	pWrite: POINTER TO BYTE;
END_VAR

pRead := pHiddenFunc + 400;
pWrite := pHiddenFunc + 4400;
HiddenPOU := TRUE;

END_FUNCTION

// MyController/Application/CheckBounds
// Implicitly generated code : DO NOT EDIT
FUNCTION CheckBounds : DINT
VAR_INPUT
	index, lower, upper: DINT;
END_VAR

// Implicitly generated code : Only an Implementation suggestion
IF  index < lower THEN
	CheckBounds := lower;
ELSIF  index > upper THEN
	CheckBounds := upper;
ELSE  
	CheckBounds := index;
END_IF

END_FUNCTION
